FUNCTION_BLOCK Axis_To_Zero
VAR_INPUT
	Flag: BOOL;
	BackZeroSpeed	:	REAL;
END_VAR
VAR_OUTPUT
END_VAR
VAR
	AxisToZero: MC_MoveAbsolute;
END_VAR

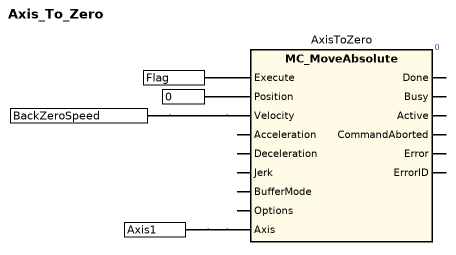
AxisToZero(Execute := Flag, Position := 0, Velocity := BackZeroSpeed, Axis := Axis1); // MC_MoveAbsolute

END_FUNCTION_BLOCK

(* stored: Version 1.1.0.1, ProductVersion 3.1.4024.12
   POU Axis_To_Zero: Id {c2527f3b-9bea-4ffc-bc68-3adc8d04dcaf}, SpecialFunc None *)
